INTERFACE ITaskStatus

METHOD Abort
END_METHOD

PROPERTY Busy : BOOL
GET
END_GET
END_PROPERTY

PROPERTY Done : BOOL
GET
END_GET
END_PROPERTY

PROPERTY Error : BOOL
GET
END_GET
END_PROPERTY

END_INTERFACE

(* stored: Version 1.1.0.1, ProductVersion 3.1.4024.5
   Itf ITaskStatus: Id {cac22837-decb-473a-90cc-a2a0eb0af979}
   Method Abort: Id {bd5ab69c-680d-4a5f-8d60-e0b5a722eb53}
   Property Busy: Id {0129cc85-1c85-4e79-9ded-86385e7537c6}
   Get Get: Id {ee3882a2-93e4-41cb-a89a-ea0695c17523}
   Property Done: Id {861ae878-400c-424e-8d3b-d7fd3d0b3027}
   Get Get: Id {64ee82f5-904a-4dc9-a108-2cc4256f4501}
   Property Error: Id {122a6517-d02a-4727-8caf-901f14e4e756}
   Get Get: Id {6535ce5e-74bd-4116-b8ac-4db07f7e5bea} *)
